TYPE JBOX_IO_Struct :
STRUCT
	SECTION : INT;
	INDEX : INT;
	CARD : STRING(10);
	TERMINAL : USINT;
	SCH_LBL : STRING(10);
	Signal : STRING(25);
	TESTER_PORT : STRING(10);
	TARGET_PORT : STRING(10);
	DESCRIPTION : STRING(255);
	LIVE_BOOL : BOOL;
	LIVE_INT : INT;
	EXPECTED_BOOL : BOOL;
	EXPECTED_INT : INT;
	RESULT : STRING(10);
END_STRUCT
END_TYPE

(* stored: Version 1.1.0.1, ProductVersion 3.1.4024.10
   DUT JBOX_IO_Struct: Id {7480ea69-84c6-4258-b51a-aa3287cb9719} *)
